// TwinCAT 3 PLC project PLC
// ProgramVersion: 3.1.4024.0
// libraries:
//   Tc2_Standard, * (Beckhoff Automation GmbH)
//   Tc2_System, * (Beckhoff Automation GmbH)
//   Tc3_Module, * (Beckhoff Automation GmbH)
// project tree:
//   10_FunctionBlocks/00_COMMON/ E_FaultLevel.TcTLEO, E_Mode.TcDUT, ST_ModuleAlarm.TcDUT
//   10_FunctionBlocks/10_CONTROL_MODE/ FB_ControlMode.TcPOU
//   10_FunctionBlocks/ ITF_ControlModules.TcIO
//   50_CONTROL_MODULE/10_VALVE/ FB_Valve.TcPOU
//   50_CONTROL_MODULE/10_VALVE/ST_ENUM/ E_ValveCommand.TcDUT, E_ValveState.TcDUT, ST_ValveConfig.TcDUT, ST_ValveStatus.TcDUT, ST_ValveErrorList.TcDUT, ST_ValveControl.TcDUT, ST_ValveSimulation.TcDUT (not stored)
//   50_CONTROL_MODULE/20_MOTOR/ FB_Motor.TcPOU
//   50_CONTROL_MODULE/20_MOTOR/ST_ENUM/ E_MotorCommand.TcDUT, E_MotorState.TcDUT (not stored), ST_MotorConfig.TcDUT, ST_MotorControl.TcDUT, ST_MotorStatus.TcDUT, ST_MotorErrorList.TcDUT, ST_MotorSimulation.TcDUT
//   50_CONTROL_MODULE/90_FUNCTIONS/ GenerateOscillation.TcPOU
//   / PlcTask.TcTTO
//   POUs/ MAIN.TcPOU
// real-time tasks:
//   TASK PlcTask: cycle T#10ms, priority 20, ADS port 350

CONFIGURATION PLC
    RESOURCE PLC ON TwinCAT3
        TASK PlcTask(INTERVAL := T#10ms, PRIORITY := 20);
        PROGRAM MAIN WITH PlcTask : MAIN;
    END_RESOURCE
END_CONFIGURATION

// ---- 10_FunctionBlocks/00_COMMON/E_FaultLevel.TcTLEO
{attribute 'qualified_only'}
{attribute 'strict'}
TYPE E_FaultLevel :
(
	DIAGNOSTIC 		:= 0,
	LOW 			:= 1,
	MEDIUM			:= 2,
	HIGH			:= 3,
	CRITICAL		:= 4
);
END_TYPE

// ---- 10_FunctionBlocks/00_COMMON/E_Mode.TcDUT
{attribute 'qualified_only'}
{attribute 'strict'}
TYPE E_Mode :
(
    MANUAL := 0,   (* Manual mode *)
    AUTO := 5,     (* Auto mode *)
	OFF := 10	   (* Off  mode *)
);
END_TYPE;

// ---- 10_FunctionBlocks/00_COMMON/ST_ModuleAlarm.TcDUT
{attribute 'OPC.UA.DA.StructuredType' := '1'}
{attribute 'OPC.UA.DA' := '1'}
{attribute 'OPC.UA.DA.Access' := '3'}
TYPE ST_ModuleAlarm :
STRUCT
	active			: BOOL;
	description		: STRING;
	level 			: E_FaultLevel;	
END_STRUCT
END_TYPE

// ---- 50_CONTROL_MODULE/10_VALVE/ST_ENUM/E_ValveCommand.TcDUT
{attribute 'qualified_only'}
{attribute 'strict'}
TYPE E_ValveCommand :
(
    CMD_OFF := 0,
    CMD_OPEN := 2,
    CMD_CLOSE := 4
);
 END_TYPE;

// ---- 50_CONTROL_MODULE/10_VALVE/ST_ENUM/E_ValveState.TcDUT
{attribute 'qualified_only'}
{attribute 'strict'}
TYPE E_ValveState :
(
    VALVE_OFF     		:= 0,
    VALVE_OPENING 		:= 1,
    VALVE_OPEN    		:= 2,
    VALVE_CLOSING 		:= 3,
    VALVE_CLOSED  		:= 4,
    VALVE_FAULT   		:= 5,
	VALVE_NEW_COMMAND   := 10
);
 END_TYPE;

// ---- 50_CONTROL_MODULE/10_VALVE/ST_ENUM/ST_ValveConfig.TcDUT
{attribute 'OPC.UA.DA.StructuredType' := '1'}
{attribute 'OPC.UA.DA' := '1'}
{attribute 'OPC.UA.DA.Access' := '3'}
TYPE ST_ValveConfig :
STRUCT
	name		   			: STRING(255);
	description				: STRING(255);
    openTimeout   			: TIME := T#15S;        (* Timeout for opening the valve *)
    closeTimeout  			: TIME := T#15S;        (* Timeout for closing the valve *)
    enableOpenFeedback   	: BOOL := FALSE; 		(* Enable feedback for open status *)
    enableCloseFeedback  	: BOOL := FALSE; 		(* Enable feedback for close status *)
END_STRUCT
END_TYPE

// ---- 50_CONTROL_MODULE/10_VALVE/ST_ENUM/ST_ValveStatus.TcDUT
{attribute 'OPC.UA.DA.StructuredType' := '1'}
{attribute 'OPC.UA.DA' := '1'}
{attribute 'OPC.UA.DA.Access' := '1'}
TYPE ST_ValveStatus :
STRUCT
    state         	: E_ValveState;        	(* Current state of the valve *)
	command         : E_ValveCommand;      	(* Current state of the valve *)
	mode   			: E_Mode;       		(* Module state: Manual, Auto, Off *)
    enabled       	: BOOL;                	(* Valve enable/disable status *)	
    elapsedTime   	: TIME;                 (* Time elapsed in current state *)
    lastOpenTime   	: TIME;                 (* Last time the valve spent opening *)
    lastCloseTime  	: TIME;                 (* Last time the valve spent closing *)
END_STRUCT
END_TYPE

// ---- 50_CONTROL_MODULE/10_VALVE/ST_ENUM/ST_ValveErrorList.TcDUT
TYPE ST_ValveErrorList :
STRUCT 
	errOpenTimeout: 		STRING	:= 'alarm open timeout';
	errLostOpenPosition: 	STRING	:= 'lost open position';
	errCloseTimeout: 		STRING	:= 'alarm closing timeout';
	errLostClosePosition: 	STRING	:= 'lost close position';
	errBothSensorOn: 		STRING	:= 'alarm both sensor on';
END_STRUCT
END_TYPE

// ---- 50_CONTROL_MODULE/10_VALVE/ST_ENUM/ST_ValveControl.TcDUT
{attribute 'OPC.UA.DA.StructuredType' := '1'}
{attribute 'OPC.UA.DA' := '1'}
{attribute 'OPC.UA.DA.Access' := '3'}
TYPE ST_ValveControl :
STRUCT
	manualOpen    			: BOOL;                 						(* OPC open command *)
    manualClose   			: BOOL;                 						(* OPC close command *)
    manualReset   			: BOOL;                 						(* OPC reset command *)
	manualModeRequest  		: E_Mode:= 	E_Mode.AUTO;       	(* OPC mode request *)
END_STRUCT
END_TYPE

// ---- 50_CONTROL_MODULE/20_MOTOR/ST_ENUM/E_MotorCommand.TcDUT
{attribute 'qualified_only'}
{attribute 'strict'}
TYPE E_MotorCommand :
(
    CMD_STOP := 0,
    CMD_MOVE_FWD := 2,
    CMD_MOVE_BCK := 4
);
 END_TYPE;

// ---- 50_CONTROL_MODULE/20_MOTOR/ST_ENUM/ST_MotorConfig.TcDUT
{attribute 'OPC.UA.DA.StructuredType' := '1'}
{attribute 'OPC.UA.DA' := '1'}
{attribute 'OPC.UA.DA.Access' := '3'}
TYPE ST_MotorConfig :
STRUCT
	name		   			: STRING(255);
	description				: STRING(255);
	manualSetpoint			: LREAL := 0.0;
    rampUpTime   			: TIME := T#15S;       
    rampDownTime  			: TIME := T#15S;       
END_STRUCT
END_TYPE

// ---- 50_CONTROL_MODULE/20_MOTOR/ST_ENUM/ST_MotorControl.TcDUT
{attribute 'OPC.UA.DA.StructuredType' := '1'}
{attribute 'OPC.UA.DA' := '1'}
{attribute 'OPC.UA.DA.Access' := '3'}
TYPE ST_MotorControl :
STRUCT
	manualStop    			: BOOL;                 
    manualMoveFwd   		: BOOL;   
	manualMoveBwd   		: BOOL;               
    manualReset   			: BOOL;                 
	manualModeRequest  		: E_Mode:= 		E_Mode.AUTO;      
END_STRUCT
END_TYPE

// ---- 50_CONTROL_MODULE/20_MOTOR/ST_ENUM/ST_MotorStatus.TcDUT
{attribute 'OPC.UA.DA.StructuredType' := '1'}
{attribute 'OPC.UA.DA' := '1'}
{attribute 'OPC.UA.DA.Access' := '1'}
TYPE ST_MotorStatus :
STRUCT
    state         	: E_MotorState;        (* Current state of the motor *)
	command        	: E_MotorCommand;      (* Current command of the motor *)
	mode   			: E_Mode;       (* Module state: Manual, Auto, Off *)
    enabled       	: BOOL;                (* Motor enable/disable status *)
	currentSpeed	: LREAL;	
	autoSetpoint	: LREAL;	
    elapsedTime   	: TIME;                 (* Time elapsed in current state *)
END_STRUCT
END_TYPE

// ---- 50_CONTROL_MODULE/20_MOTOR/ST_ENUM/ST_MotorErrorList.TcDUT
TYPE ST_MotorErrorList :
STRUCT 
END_STRUCT
END_TYPE

// ---- 50_CONTROL_MODULE/20_MOTOR/ST_ENUM/ST_MotorSimulation.TcDUT
{attribute 'OPC.UA.DA.StructuredType' := '1'}
{attribute 'OPC.UA.DA' := '1'}
TYPE ST_MotorSimulation :
STRUCT
	simEnable				: BOOL;
	{attribute 'OPC.UA.DA' := '0'}
	T_RampUpTime			: TON;
	{attribute 'OPC.UA.DA' := '0'}
	T_RampDownTime			: TON;
END_STRUCT
END_TYPE

// ---- 10_FunctionBlocks/ITF_ControlModules.TcIO
INTERFACE ITF_ControlModules

METHOD M_RaiseFault : BOOL
VAR_INPUT
	description		: STRING;
	level 			: E_FaultLevel;
END_VAR
END_METHOD

METHOD M_ResetFault : BOOL
VAR_INPUT
END_VAR
END_METHOD

PROPERTY P_mode : E_Mode;
GET
END_GET
END_PROPERTY

END_INTERFACE

// ---- POUs/MAIN.TcPOU
PROGRAM MAIN
VAR
	valve1			: FB_Valve;
	valve2			: FB_Valve;
	valve3			: FB_Valve;
	
	motor1			: FB_Motor;
	
	step		: INT;
	{attribute 'OPC.UA.DA' := '1'}
	startCycle 	: BOOL;
	auto		: BOOL;
	cycleTimer	: TON;
END_VAR

CASE step OF 
	// START
	0: 
	IF startCycle THEN
		step := 5;
	END_IF
	
	// REQUEST AUTO
	5:
	step := 10;
	auto := TRUE;
	
	// OPEN VALVE 1
	10:
	IF 	valve1.P_mode = E_Mode.AUTO AND
		valve2.P_mode = E_Mode.AUTO AND
		valve3.P_mode = E_Mode.AUTO THEN
		valve1.M_Open_Auto();
		step := 15;
	END_IF
	
	// OPEN VALVE 2,3
	15: 
	IF 	valve1.P_state = E_ValveState.VALVE_OPEN THEN 
		valve2.M_Open_Auto();
		valve3.M_Open_Auto();
		step := 20;
	END_IF
	
	// PAUSE 
	20: 
	IF 	valve2.P_state = E_ValveState.VALVE_OPEN AND
		valve3.P_state = E_ValveState.VALVE_OPEN THEN 
		step := 21;
	END_IF
	
	//  CLOSE VALVE 2
	21:
	cycleTimer(IN:= TRUE, PT:= T#3S);
	IF 	cycleTimer.Q THEN
		cycleTimer(IN:= FALSE);
		valve2.M_CloseAuto();
		step := 25;
	END_IF
		
	// CLOSE VALVE 3
	25: 
	IF 	valve2.P_state = E_ValveState.VALVE_CLOSED THEN
		valve3.M_CloseAuto();
		step := 30;
	END_IF
	// CLOSE VALVE 1
	30: 
	IF 	valve3.P_state = E_ValveState.VALVE_CLOSED THEN
		valve1.M_CloseAuto();
		step := 35;
	END_IF
	35: 
	IF 	valve1.P_state = E_ValveState.VALVE_CLOSED THEN
		auto := FALSE;
		step := 40;
	END_IF
	40: 
	cycleTimer(IN:= TRUE, PT:= T#2S);
	IF 	cycleTimer.Q THEN
		cycleTimer(IN:= FALSE);
		step := 0;
	END_IF
	
	
END_CASE

valve1(ib_enable:=TRUE, ib_auto:= auto  );
valve2(ib_enable:=TRUE, ib_auto:= auto  );
valve3(ib_enable:=TRUE, ib_auto:= auto  );
valve1.P_simulation := TRUE;
valve2.P_simulation := TRUE;
valve3.P_simulation := TRUE;

motor1(ib_enable:=TRUE, ib_auto:= auto  );
motor1.P_simulation := TRUE;

END_PROGRAM

// ---- 50_CONTROL_MODULE/10_VALVE/FB_Valve.TcPOU
FUNCTION_BLOCK FB_Valve EXTENDS FB_ControlMode
VAR_INPUT
	ib_openFeedback			: BOOL;
	ib_closeFeedback		: BOOL;	
END_VAR

VAR_OUTPUT
    ob_openCommand   		:  BOOL;  
	ob_closeCommand   		:  BOOL;       
END_VAR

VAR
	// OPC VARIABLES
	status 		   			: ST_ValveStatus  ;
	control					: ST_ValveControl;
	sim						: ST_ValveSimulation;
	
	// FB VARIABLES
	ton_openTime			: TON;
	ton_closeTime			: TON;
	startOpen				: BOOL;
	startClose				: BOOL;
    ton_ElapsedTime   		: TON;                	(* Timer for monitor current operation *)
	startMovement			: BOOL;
	error 					: ST_ValveErrorList;
	openFeedback			: BOOL;
	closeFeedback			: BOOL;
END_VAR

VAR PERSISTENT
	config       			: ST_ValveConfig;      		(* Valve configuration parameters *)
END_VAR

// MODULE STATE LOGIC
SUPER^.requestMode := control.manualModeRequest;
SUPER^();  
CASE mode OF 
	
	E_Mode.OFF:
		M_Private_Off();
	
	E_Mode.MANUAL:
		// manual logic:
		;
	E_Mode.AUTO:
		// auto logic:
		;	
END_CASE


// manual control logic
M_Private_ManualControl();

// feedback simulation logic
IF sim.simEnable THEN
	M_Simulation();
END_IF

openFeedback := ib_openFeedback OR sim.simOpenFeedback;
closeFeedback := ib_closeFeedback OR sim.simCloseFeedback;

// MAIN LOGIC
CASE status.command OF		
	E_ValveCommand.CMD_OFF:
		ob_OpenCommand := FALSE;
		ob_CloseCommand:= FALSE;
		startMovement := FALSE;
		

	E_ValveCommand.CMD_CLOSE:
		ob_OpenCommand := FALSE;
		ob_CloseCommand:= TRUE;
		
		CASE status.state OF
		
		E_ValveState.VALVE_NEW_COMMAND: 
			status.state := E_ValveState.VALVE_CLOSING;
			
		E_ValveState.VALVE_CLOSING: 
			IF CloseFeedback OR NOT config.enableCloseFeedback THEN
				status.state:= E_ValveState.VALVE_CLOSED;
			ELSIF ton_ElapsedTime.et >= config.closeTimeout THEN
				(* Timeout occurred *)
				status.state:= E_ValveState.VALVE_FAULT;
				M_RaiseFault(description := error.errCloseTimeout, level := E_FaultLevel.HIGH);
			END_IF
		E_ValveState.VALVE_CLOSED: 
			startMovement := FALSE;
			IF NOT CloseFeedback AND config.enableCloseFeedback THEN
				status.state:= E_ValveState.VALVE_FAULT;
				M_RaiseFault(description := error.errLostClosePosition, level := E_FaultLevel.HIGH);
			END_IF
		END_CASE
		
		
	E_ValveCommand.CMD_OPEN:
		ob_OpenCommand := TRUE;
		ob_CloseCommand:= FALSE;
		
		CASE status.state OF
		
		E_ValveState.VALVE_NEW_COMMAND: 
			status.state := E_ValveState.VALVE_OPENING;
			
		E_ValveState.VALVE_OPENING: 
			IF OpenFeedback OR NOT config.enableOpenFeedback THEN
				status.state:= E_ValveState.VALVE_OPEN;
			ELSIF ton_ElapsedTime.et >= config.openTimeout THEN
				(* Timeout occurred *)
				status.state:= E_ValveState.VALVE_FAULT;
				M_RaiseFault(description := error.errOpenTimeout, level := E_FaultLevel.HIGH);
			END_IF
		E_ValveState.VALVE_OPEN: 
			startMovement := FALSE;
			IF NOT openFeedback AND config.enableOpenFeedback THEN
				status.state:= E_ValveState.VALVE_FAULT;
				M_RaiseFault(description := error.errLostOpenPosition, level := E_FaultLevel.HIGH);
			END_IF
		END_CASE
		
END_CASE

// OPC VARIABLES
status.mode := mode;
status.enabled := ib_enable;

// TIMER LOGIC
ton_ElapsedTime(IN:=startMovement, PT:=T#2147483647MS );
IF startMovement THEN
	status.elapsedTime := ton_ElapsedTime.ET;
END_IF

ton_openTime(IN:=startOpen, 	PT:=T#2147483647MS );
IF startOpen AND ( openFeedback OR NOT config.enableOpenFeedback ) THEN
	startOpen := FALSE;
	status.lastOpenTime := ton_openTime.ET ;
END_IF

ton_closeTime(IN:=startClose, 	PT:=T#2147483647MS );
IF startClose AND ( closeFeedback OR NOT config.enableOpenFeedback ) THEN
	startClose := FALSE;
	status.lastCloseTime := ton_closeTime.ET ;
END_IF

METHOD M_CloseAuto : BOOL
IF status.mode = E_Mode.AUTO THEN
	M_Private_CloseValve();
END_IF
END_METHOD

METHOD M_Open_Auto : BOOL
IF status.mode = E_Mode.AUTO THEN
	M_Private_OpenValve();
END_IF
END_METHOD

METHOD PRIVATE M_Private_CloseValve : BOOL
status.state 	:= E_ValveState.VALVE_NEW_COMMAND;
status.command 	:= E_ValveCommand.CMD_CLOSE;
startMovement 	:= TRUE;
startClose 		:= TRUE;
status.elapsedTime := T#0S;
M_resetFault();
END_METHOD

METHOD PRIVATE M_Private_ManualControl : BOOL
IF status.mode = E_Mode.MANUAL THEN
	IF control.ManualOpen THEN 
		control.ManualOpen := FALSE;
		M_Private_OpenValve();
	ELSIF control.ManualClose THEN 
		control.ManualClose := FALSE;
		M_Private_CloseValve();
	END_IF
ELSE
	control.ManualOpen := FALSE;
	control.ManualClose := FALSE;
END_IF

IF control.ManualReset THEN 
	control.ManualReset := FALSE;
	M_resetFault();
	status.state := E_ValveState.VALVE_NEW_COMMAND;
END_IF
END_METHOD

METHOD PRIVATE M_Private_Off : BOOL
status.state := E_ValveState.VALVE_OFF;
status.command := E_ValveCommand.CMD_OFF;
status.elapsedTime := T#0S;
M_resetFault();
END_METHOD

METHOD PRIVATE M_Private_OpenValve : BOOL
status.state 	:= E_ValveState.VALVE_NEW_COMMAND;
status.command 	:= E_ValveCommand.CMD_OPEN;
startMovement 	:= TRUE;
startOpen	  	:= TRUE;
status.elapsedTime := T#0S;
M_resetFault();
END_METHOD

METHOD M_Simulation : BOOL
VAR_INPUT
END_VAR
sim.T_CloseFeedback(IN:= status.command=E_ValveCommand.CMD_CLOSE, PT := T#5S, Q=> sim.simCloseFeedback);
sim.T_OpenFeedback(IN:= status.command=E_ValveCommand.CMD_OPEN, PT := T#5S, Q=> sim.simOpenFeedback);
END_METHOD

PROPERTY P_simulation : REFERENCE TO BOOL
GET
P_Simulation REF= sim.simEnable;
END_GET
END_PROPERTY

PROPERTY P_state : E_ValveState
GET
P_state:=status.state;
END_GET
END_PROPERTY

END_FUNCTION_BLOCK

// ---- 10_FunctionBlocks/10_CONTROL_MODE/FB_ControlMode.TcPOU
FUNCTION_BLOCK FB_ControlMode IMPLEMENTS ITF_ControlModules
VAR_INPUT
    ib_enable      	: BOOL;           // Input to enable the module
    ib_auto        	: BOOL;           // Input to request automatic mode
END_VAR

VAR 
	fault			: ST_ModuleAlarm;  // OPC fault variable
	mode 			: E_Mode;
	requestMode		: E_Mode;
END_VAR

// NOT ENABLE BY PLC
IF NOT ib_enable THEN
	(* If not enabled by PLC , set the module to OFF *)
	mode := E_Mode.OFF;
	M_RaiseFault(description := 'Module disabled', level := E_FaultLevel.DIAGNOSTIC);
// PARENT AUTO REQUEST	
ELSIF ib_auto THEN 
	(* module already in auto *) 
	IF mode = E_Mode.AUTO THEN
		requestMode := E_Mode.AUTO;
		M_RaiseFault(description := 'Controlled by parent system', level := E_FaultLevel.DIAGNOSTIC);
	(* wait to release manual or off mode *)
	ELSIF requestMode = E_Mode.AUTO THEN
		mode := E_Mode.AUTO;
	(* info the parent is requesting auto mode *)
	ELSE
		M_RaiseFault(description := 'Request auto mode from parent system', level := E_FaultLevel.DIAGNOSTIC);
	END_IF
ELSE
	// Manual mode - state is controlled by the HMI input
	mode := requestMode;
	
	// Handle OFF state separately
	IF mode = E_Mode.OFF THEN
		M_RaiseFault(description := 'Module set to OFF by operator', level := E_FaultLevel.DIAGNOSTIC);
	END_IF
END_IF

METHOD M_RaiseFault : BOOL
VAR_INPUT
	description	: STRING;
	level	: E_FaultLevel;
END_VAR
fault.active 		:= TRUE ;
fault.description 	:= description ;
fault.level			:= level;
END_METHOD

METHOD M_ResetFault : BOOL
fault.active 		:= FALSE ;
fault.description 	:= '' ;
fault.level			:= E_FaultLevel.DIAGNOSTIC;
END_METHOD

PROPERTY P_mode : E_Mode;
GET
P_mode := mode;
END_GET
END_PROPERTY

END_FUNCTION_BLOCK

// ---- 50_CONTROL_MODULE/20_MOTOR/FB_Motor.TcPOU
FUNCTION_BLOCK FB_Motor EXTENDS FB_ControlMode
VAR_INPUT
END_VAR

VAR_OUTPUT      
END_VAR

VAR
	// OPC VARIABLES
	status 		   			: ST_MotorStatus  ;
	control					: ST_MotorControl;
	sim						: ST_MotorSimulation;
	
	// FB VARIABLES
	actualSpeed				: LREAL;
	setpoint				: LREAL;
    ton_ElapsedTime   		: TON;                	(* Timer for monitor current operation *)
	error 					: ST_MotorErrorList;
	
	rRand 		: LREAL ;
	randGen		: DRAND ;
	randValue	: LREAL;
END_VAR

VAR PERSISTENT
	config       			: ST_MotorConfig;      		(* Valve configuration parameters *)
END_VAR

// MODULE STATE LOGIC
SUPER^.requestMode := control.manualModeRequest;
SUPER^();  
CASE mode OF 
	
	E_Mode.OFF:
		M_Private_Off();
	
	E_Mode.MANUAL:
		// manual logic:
		;
	E_Mode.AUTO:
		// auto logic:
		;	
END_CASE

// manual mode logic
M_Private_ManualControl();

// feedback simulation logic
IF sim.simEnable THEN
	M_Simulation();
END_IF

// OPC VARIABLES
status.mode 	:= mode;
status.enabled 	:= ib_enable;
status.currentSpeed 	:= actualSpeed;
// TIMER LOGIC
ton_ElapsedTime(IN:=FALSE, PT:=T#2147483647MS );
IF FALSE THEN
	status.elapsedTime := ton_ElapsedTime.ET;
END_IF

METHOD PRIVATE M_moveBck : BOOL
VAR_INPUT
	ir_setpoint : LREAL := 0.0;
END_VAR
status.state 			:= E_MotorState.MOVING_BCK;
status.command 		:= E_MotorCommand.CMD_MOVE_BCK;
setpoint 			:= ir_setpoint;
status.elapsedTime 	:= T#0S;
M_resetFault();
END_METHOD

METHOD M_moveBck_Auto : BOOL
VAR_INPUT
	ir_setpoint : LREAL := 0.0;
END_VAR
IF status.mode = E_Mode.AUTO THEN
	M_MoveBck(ir_setpoint:= ir_setpoint);
END_IF
END_METHOD

METHOD PRIVATE M_moveFwd : BOOL
VAR_INPUT
	ir_setpoint : LREAL := 0.0;
END_VAR
status.state 			:= E_MotorState.MOVING_FWD;
status.command 		:= E_MotorCommand.CMD_MOVE_FWD;
setpoint 			:= ir_setpoint;
status.elapsedTime 	:= T#0S;
M_resetFault();
END_METHOD

METHOD M_moveFwd_Auto : BOOL
VAR_INPUT
	ir_setpoint : LREAL := 0.0;
END_VAR
IF status.mode = E_Mode.AUTO THEN
	M_MoveFwd(ir_setpoint:= ir_setpoint);
END_IF
END_METHOD

METHOD PRIVATE M_Private_ManualControl : BOOL
IF status.mode = E_Mode.MANUAL THEN
	IF control.manualMoveFwd THEN 
		control.manualMoveFwd := FALSE;
		M_moveFwd(ir_setpoint := config.manualSetpoint);
	ELSIF control.manualMoveBwd THEN 
		control.manualMoveBwd := FALSE;
		M_moveBck(ir_setpoint := config.manualSetpoint);
	ELSIF control.manualStop THEN 
		control.manualStop := FALSE;
		M_stop();
	END_IF
ELSE
	control.manualMoveFwd := FALSE;
	control.manualMoveBwd := FALSE;
	control.manualStop := FALSE;
END_IF

IF control.ManualReset THEN 
	control.ManualReset := FALSE;
	M_resetFault();
END_IF
END_METHOD

METHOD PRIVATE M_Private_Off : BOOL
status.state := E_MotorState.OFF;
status.command := E_MotorCommand.CMD_STOP;
status.elapsedTime := T#0S;
M_resetFault();
END_METHOD

METHOD M_Simulation : BOOL
VAR
END_VAR

VAR CONSTANT
    rRampRateUp 		: LREAL := 0.1;   // Speed increment rate during ramp-up
    rRampRateDown 		: LREAL := 0.5; // Speed decrement rate during ramp-down
    rOscillationRange 	: LREAL := 4; // Range for oscillation around setpoint
END_VAR
randGen(seed:= 0, Num=>randValue);
rRand := (randValue - 0.5) * rOscillationRange ; // Generates random value between -rOscillationRange and +rOscillationRange

// Main Logic
IF status.command = E_MotorCommand.CMD_MOVE_FWD OR status.command = E_MotorCommand.CMD_MOVE_BCK THEN
    // Ramp-up to the setpoint
    IF actualSpeed < setpoint THEN
        actualSpeed := actualSpeed + rRampRateUp;
    ELSE
        actualSpeed := setpoint - rRampRateUp;
    END_IF

ELSIF status.command = E_MotorCommand.CMD_STOP THEN
    // Ramp-down to zero
    IF actualSpeed > 0 THEN
        actualSpeed := actualSpeed - rRampRateDown;
    ELSIF actualSpeed < 0 THEN
        actualSpeed := 0;
    END_IF

END_IF

// Simulate oscillation when running
IF status.command = E_MotorCommand.CMD_MOVE_BCK OR status.command = E_MotorCommand.CMD_MOVE_FWD THEN
    actualSpeed := actualSpeed + rRand;
ELSE
    actualSpeed := actualSpeed;
END_IF
END_METHOD

METHOD PRIVATE M_stop : BOOL
status.state 	:= E_MotorState.STOP;
status.command := E_MotorCommand.CMD_STOP;
status.elapsedTime := T#0S;
M_resetFault();
END_METHOD

METHOD M_stopAuto : BOOL
IF status.mode = E_Mode.AUTO THEN
	M_stop();
END_IF
END_METHOD

PROPERTY P_simulation : REFERENCE TO BOOL;
GET
P_simulation REF= sim.simEnable;
END_GET
END_PROPERTY

PROPERTY P_state : E_MotorState
GET
P_state:=status.state;
END_GET
END_PROPERTY

END_FUNCTION_BLOCK

// ---- 50_CONTROL_MODULE/90_FUNCTIONS/GenerateOscillation.TcPOU
FUNCTION GenerateOscillation : REAL
VAR_INPUT
	rRand: REAL;
END_VAR
VAR
END_VAR

rRand := (RAND() - 0.5) * rOscillationRange * 2; // Generates random value between -rOscillationRange and +rOscillationRange
    GenerateOscillation := rRand;

END_FUNCTION
